// TIA Portal project "FactoryIO_Template_S7-1200_V15_V18_2" (V18)
// Vorlageprojekt für das Buch mit Zielsystem S7-1200

(* hardware
DEVICE "S7-1200-Station_1"  S7-1200 Station
   slot 0: "Baugruppenträger_0"  Rack  V1.0
   slot 1: "PLC_1"  CPU 1214C DC/DC/Rly  6ES7 214-1HG40-0XB0  V4.6
*)

// ===== PLC "PLC_1"  CPU 1214C DC/DC/Rly =====

VAR_GLOBAL   // PLC tag table "Standard-Variablentabelle"
   "motor_main" AT %A0.0 : Bool;
   "Start_but" AT %E0.0 : Bool;
   "Stop_but" AT %E0.1 : Bool;
   "Start_mem" AT %M0.0 : Bool;
   "Emergency_stop" AT %M10.5 : Bool;
   "palet_sensor" AT %I0.3 : Bool;
   "down_sensor" AT %I0.4 : Bool;
   "transfer_motor_mem" AT %M1.1 : Bool;
   "upload_sensor" AT %I0.5 : Bool;
   "right_motor" AT %Q0.2 : Bool;
   "up_sensor" AT %I0.6 : Bool;
   "left_motor" AT %Q0.3 : Bool;
   "transfer_motor" AT %Q0.4 : Bool;
   "motor_stop" AT %M1.0 : Bool;
   "right_motor_mem" AT %M1.2 : Bool;
   "motor_main_right" AT %Q0.6 : Bool;
   "motor_main_left" AT %Q0.7 : Bool;
   "right_transfer" AT %Q1.0 : Bool;
   "left_transfer" AT %Q1.1 : Bool;
   "right_transfer_mem" AT %M2.0 : Bool;
   "left_transfer_mem" AT %M2.1 : Bool;
   "left_transfer_stop_mem" AT %M2.2 : Bool;
   "Tag_2" AT %I2.0 : Bool;
   "left_transfer_sensor" AT %I1.3 : Bool;
   "right_transfer_sensor" AT %I1.4 : Bool;
   "right_transfer_stop_mem" AT %M2.3 : Bool;
   "reset_but" AT %I1.7 : Bool;
   "Tag_1" AT %M10.0 : Bool;
   "upload_sensor_mem" AT %M10.1 : Bool;
   "warning_lamb" AT %Q1.7 : Bool;
   "Tag_3" AT %M11.0 : Bool;
END_VAR

// folder: System blocks/Program resources

DATA_BLOCK "timer1"   // DB1
{ S7_Optimized_Access := 'TRUE' }
AUTHOR : Simatic
FAMILY : IEC
NAME : IEC_TMR
VERSION : 1.0
// stored: InstanceOfName IEC_TIMER
"IEC_TIMER"
BEGIN
END_DATA_BLOCK

DATA_BLOCK "timer10"   // DB2
{ S7_Optimized_Access := 'TRUE' }
AUTHOR : Simatic
FAMILY : IEC
NAME : IEC_TMR
VERSION : 1.0
// stored: InstanceOfName IEC_TIMER
"IEC_TIMER"
BEGIN
END_DATA_BLOCK

DATA_BLOCK "timer3"   // DB3
{ S7_Optimized_Access := 'TRUE' }
AUTHOR : Simatic
FAMILY : IEC
NAME : IEC_TMR
VERSION : 1.0
// stored: InstanceOfName IEC_TIMER
"IEC_TIMER"
BEGIN
END_DATA_BLOCK

DATA_BLOCK "timer7"   // DB4
{ S7_Optimized_Access := 'TRUE' }
AUTHOR : Simatic
FAMILY : IEC
NAME : IEC_TMR
VERSION : 1.0
// stored: InstanceOfName IEC_TIMER
"IEC_TIMER"
BEGIN
END_DATA_BLOCK

DATA_BLOCK "timer6"   // DB6
{ S7_Optimized_Access := 'TRUE' }
AUTHOR : Simatic
FAMILY : IEC
NAME : IEC_TMR
VERSION : 1.0
// stored: InstanceOfName IEC_TIMER
"IEC_TIMER"
BEGIN
END_DATA_BLOCK

DATA_BLOCK "timer8"   // DB7
{ S7_Optimized_Access := 'TRUE' }
AUTHOR : Simatic
FAMILY : IEC
NAME : IEC_TMR
VERSION : 1.0
// stored: InstanceOfName IEC_TIMER
"IEC_TIMER"
BEGIN
END_DATA_BLOCK

DATA_BLOCK "timer9"   // DB8
{ S7_Optimized_Access := 'TRUE' }
AUTHOR : Simatic
FAMILY : IEC
NAME : IEC_TMR
VERSION : 1.0
// stored: InstanceOfName IEC_TIMER
"IEC_TIMER"
BEGIN
END_DATA_BLOCK

// folder: (top level)

FUNCTION "MHJ-PLC-Lab-Function-S71200" : Void   // FC9000, SCL
{ S7_Optimized_Access := 'TRUE' }
VERSION : 0.1
   VAR_TEMP
      rdTimeReturn : Int;
      outputTime : DTL;
      SyncVal : Byte;
      forVal : Int;
      forVal_2 : Int;
      Value : Byte;
   END_VAR
   VAR CONSTANT
      CompVal : Byte := 16#34;
      Value_01 : Byte := 16#11;
      Value_01_DW : DWord := 16#A165_D992;
      Value_02_DW : DWord := 16#58BE_4401;
   END_VAR
BEGIN

   #Value:=PEEK(area := 16#82,
        dbNumber := 0,
        byteOffset := 511);
   #Value := #Value + 1;

   POKE(area := 16#82,
        dbNumber := 0,
        byteOffset := 511,
        value := #Value);

   POKE(area:=16#81,
        dbNumber:=0,
        byteOffset:=1016,
        value:=#Value_01_DW);
   POKE(area := 16#81,
        dbNumber := 0,
        byteOffset := 1020,
        value := #Value_02_DW);

   POKE(area := 16#81,
        dbNumber := 0,
        byteOffset := 511,
        value := B#16#00);

   FOR #forVal := 0 TO 120 DO
       FOR #forVal_2:=0 TO 10 DO
           #rdTimeReturn:=RD_SYS_T(#outputTime);
           #rdTimeReturn := WR_SYS_T(#outputTime);
           #rdTimeReturn := RD_SYS_T(#outputTime);
           #rdTimeReturn := WR_SYS_T(#outputTime);
       END_FOR;
       #SyncVal:= PEEK(area := 16#81,
                      dbNumber := 0,
                      byteOffset := 511);
       IF #SyncVal = #CompVal THEN
          GOTO M_1;
       END_IF;
   END_FOR;
   RETURN;

   M_1:
   POKE(area := 16#81,
        dbNumber := 0,
        byteOffset := 511,
        value := B#16#0);
END_FUNCTION

ORGANIZATION_BLOCK "Main"   // OB1, LAD, ProgramCycle
TITLE = "Main Program Sweep (Cycle)"
{ S7_Optimized_Access := 'TRUE' }
VERSION : 0.1
   VAR_INPUT
      Initial_Call : Bool;   // Initial call of this OB
      Remanence : Bool;   // =True, if remanent data are available
   END_VAR
   VAR_TEMP   // added for the SCL form of the ladder/FBD networks
      _w1 : Bool;
      _w2 : Bool;
   END_VAR
BEGIN

REGION Network 1: Konnektierungsbaustein für PLC-Lab
   // Im Netzwerk 1 wird der Konnektierungsbaustein für PLC-Lab aufgerufen.
   // Dieser Aufruf darf nicht entfernt werden!
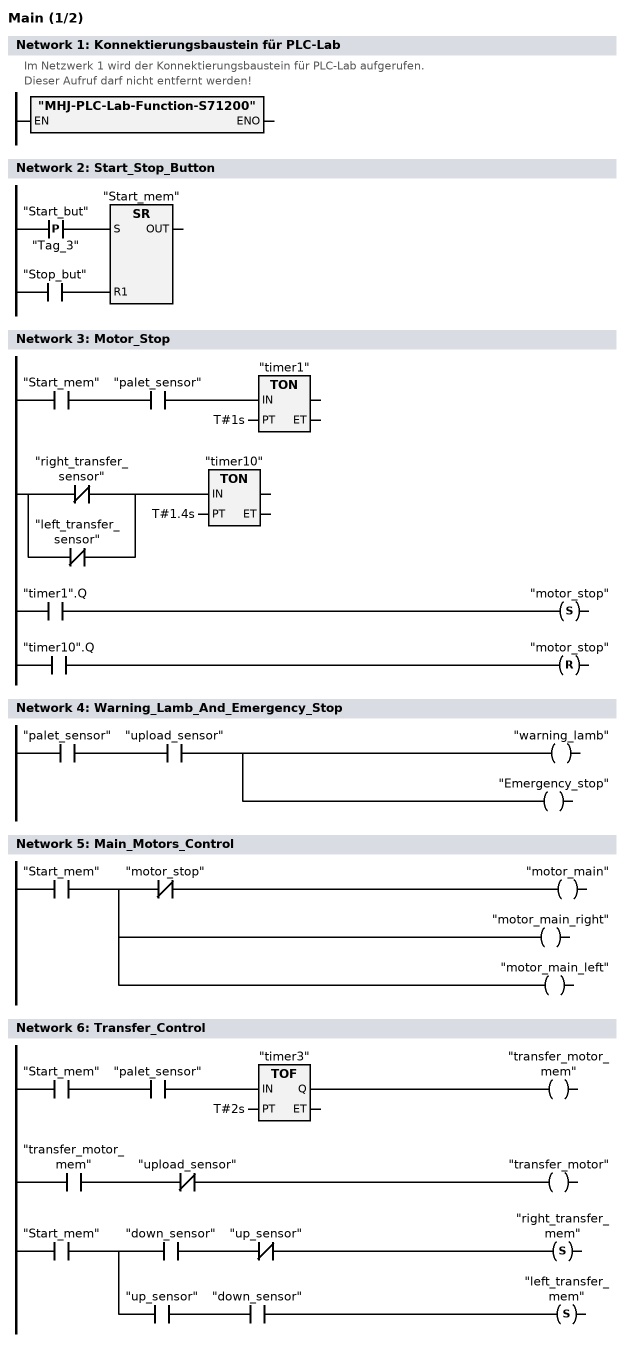
   RUNG wire#powerrail
      "MHJ-PLC-Lab-Function-S71200"()
   END_RUNG
   // the same network as SCL:
   "MHJ-PLC-Lab-Function-S71200"();
END_REGION

REGION Network 2: Start_Stop_Button
   RUNG wire#powerrail
      P_Contact(operand := "Start_but", bit := "Tag_3")
      S_SR(operand := "Start_mem", r1 := wire#w1)
   END_RUNG
   RUNG wire#powerrail
      Contact( "Stop_but" )
   END_RUNG wire#w1
   // the same network as SCL:
   #_w1 := "Start_but" AND NOT "Tag_3";   // rising edge of "Start_but"
   "Tag_3" := "Start_but";
   IF #_w1 THEN
       "Start_mem" := TRUE;   // SR flip-flop
   END_IF;
   IF "Stop_but" THEN "Start_mem" := FALSE; END_IF;
END_REGION

REGION Network 3: Motor_Stop
   "timer1".TON(IN := "Start_mem" AND "palet_sensor", PT := T#1s);
   "timer10".TON(IN := NOT "right_transfer_sensor" OR NOT "left_transfer_sensor", PT := T#1.4s);
   IF "timer1".Q THEN "motor_stop" := TRUE; END_IF;
   IF "timer10".Q THEN "motor_stop" := FALSE; END_IF;
END_REGION

REGION Network 4: Warning_Lamb_And_Emergency_Stop
   RUNG wire#powerrail
      Contact( "palet_sensor" )
      Contact( "upload_sensor" )
      wire#w1
      Coil( "warning_lamb" )
   END_RUNG
   RUNG wire#w1
      Coil( "Emergency_stop" )
   END_RUNG
   // the same network as SCL:
   "warning_lamb" := "palet_sensor" AND "upload_sensor";
   "Emergency_stop" := "warning_lamb";
END_REGION

REGION Network 5: Main_Motors_Control
   RUNG wire#powerrail
      Contact( "Start_mem" )
      wire#w1
      I_Contact( "motor_stop" )
      Coil( "motor_main" )
   END_RUNG
   RUNG wire#w1
      Coil( "motor_main_right" )
   END_RUNG
   RUNG wire#w1
      Coil( "motor_main_left" )
   END_RUNG
   // the same network as SCL:
   "motor_main" := "Start_mem" AND NOT "motor_stop";
   "motor_main_right" := "Start_mem";
   "motor_main_left" := "Start_mem";
END_REGION

REGION Network 6: Transfer_Control
   "timer3".TOF(IN := "Start_mem" AND "palet_sensor", PT := T#2s);
   "transfer_motor_mem" := "timer3".Q;
   "transfer_motor" := "transfer_motor_mem" AND NOT "upload_sensor";
   IF "Start_mem" AND "down_sensor" AND NOT "up_sensor" THEN "right_transfer_mem" := TRUE; END_IF;
   IF "Start_mem" AND "up_sensor" AND "down_sensor" THEN "left_transfer_mem" := TRUE; END_IF;
END_REGION

REGION Network 7
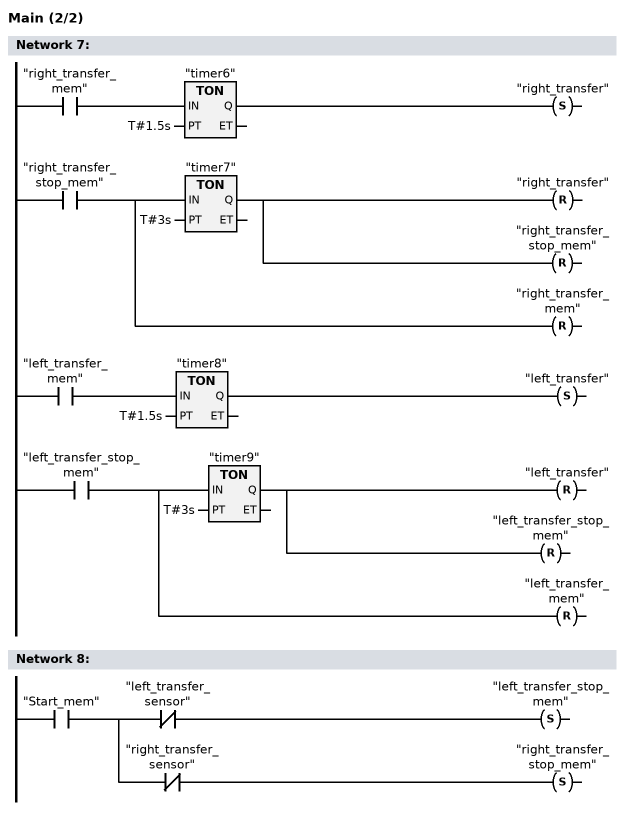
   "timer6".TON(IN := "right_transfer_mem", PT := T#1.5s);
   IF "timer6".Q THEN "right_transfer" := TRUE; END_IF;
   "timer7".TON(IN := "right_transfer_stop_mem", PT := T#3s);
   IF "timer7".Q THEN "right_transfer" := FALSE; END_IF;
   #_w1 := "right_transfer_stop_mem";
   IF "timer7".Q THEN "right_transfer_stop_mem" := FALSE; END_IF;
   IF #_w1 THEN "right_transfer_mem" := FALSE; END_IF;
   "timer8".TON(IN := "left_transfer_mem", PT := T#1.5s);
   IF "timer8".Q THEN "left_transfer" := TRUE; END_IF;
   "timer9".TON(IN := "left_transfer_stop_mem", PT := T#3s);
   IF "timer9".Q THEN "left_transfer" := FALSE; END_IF;
   #_w2 := "left_transfer_stop_mem";
   IF "timer9".Q THEN "left_transfer_stop_mem" := FALSE; END_IF;
   IF #_w2 THEN "left_transfer_mem" := FALSE; END_IF;
END_REGION

REGION Network 8
   RUNG wire#powerrail
      Contact( "Start_mem" )
      wire#w1
      I_Contact( "left_transfer_sensor" )
      S_Coil( "left_transfer_stop_mem" )
   END_RUNG
   RUNG wire#w1
      I_Contact( "right_transfer_sensor" )
      S_Coil( "right_transfer_stop_mem" )
   END_RUNG
   // the same network as SCL:
   IF "Start_mem" AND NOT "left_transfer_sensor" THEN "left_transfer_stop_mem" := TRUE; END_IF;
   IF "Start_mem" AND NOT "right_transfer_sensor" THEN "right_transfer_stop_mem" := TRUE; END_IF;
END_REGION
END_ORGANIZATION_BLOCK